TYPE UnwindCmd_Typ :
STRUCT
	JogFwd:BOOL;
	JogBack:BOOL;
	JogSFwdSlow:BOOL;
	JogBackdSlow:BOOL;
	JogDancerFill:BOOL;	
END_STRUCT
END_TYPE

(* stored: Version 1.1.0.1, ProductVersion 3.1.4024.3
   DUT UnwindCmd_Typ: Id {f00549d1-2b35-42df-97ed-155f8899630d} *)
